# EPICS alarm handler configuration: mps_database/bareTest/alarms/areas/mpln_ltus_mp01.alhConfig
GROUP NULL MPLN:LTUS:MP01:1
$ALIAS MPS Link Node 203
$GUIDANCE
LTUH MPS
   Group Name: MPLN:LTUS:MP01:1
   Summary PV:  MPLN:LTUS:MP01:1:STATSUMY
$END
CHANNEL  MPLN:LTUS:MP01:1    MPLN:LTUS:MP01:1:MPS_EN_RBV		-----
CHANNEL  MPLN:LTUS:MP01:1    MPLN:LTUS:MP01:1:LC1_MODE_RBV		-----
